// TwinCAT 3 PLC project PLC
// ProgramVersion: 3.1.4026.19
// CompilerDefines: VISU_USEPROPERTYINFO
// libraries:
//   Tc2_MC2, * (Beckhoff Automation GmbH)
//   Tc2_Standard, * (Beckhoff Automation GmbH)
//   Tc2_System, * (Beckhoff Automation GmbH)
//   VisuDialogs, * (System)
// project tree:
//   / GlobalTextList.TcGTLO, PlcTask.TcTTO, Visualization Manager.TcVMO (not stored)
//   POUs/ MAIN.TcPOU
//   VISUs/ HomeScreen.TcVIS

CONFIGURATION PLC
    RESOURCE PLC ON TwinCAT3
        TASK PlcTask(INTERVAL := T#10ms, PRIORITY := 20);
        PROGRAM MAIN WITH PlcTask : MAIN;
    END_RESOURCE
END_CONFIGURATION

// ---- POUs/MAIN.TcPOU
PROGRAM MAIN
VAR
	axisVirtualMotor : AXIS_REF;
	fbPower : MC_Power;
	fbMoveAbs : MC_MoveAbsolute;
	bEnable : BOOL;
	bMoveStart : BOOL;
	fTargetLocation : LREAL := 250.5;
	fLocation : LREAL;
END_VAR

fbPower(
	Axis := axisVirtualMotor,
	Enable := bEnable,
	Enable_Positive := bEnable,
	Enable_Negative := bEnable,
	Override := 100.0
);

fbMoveAbs(
	Axis := axisVirtualMotor,
	Execute := bMoveStart,
	Position := fTargetLocation,
	Velocity := 100.0,
	Acceleration := 100.0,
	Deceleration := 100.0,
	Jerk := 100.0
);

fLocation := axisVirtualMotor.NcToPlc.ActPos;

END_PROGRAM

// ---- GlobalTextList.TcGTLO
TEXTLIST GlobalTextList
  621 = 'Location: %.2f mm'
  700 = 'Power Off'
  717 = 'Power On'
  63 = 'Start to Move'
  985 = 'Target: %.2f mm'
END_TEXTLIST

// ---- VISUs/HomeScreen.TcVIS
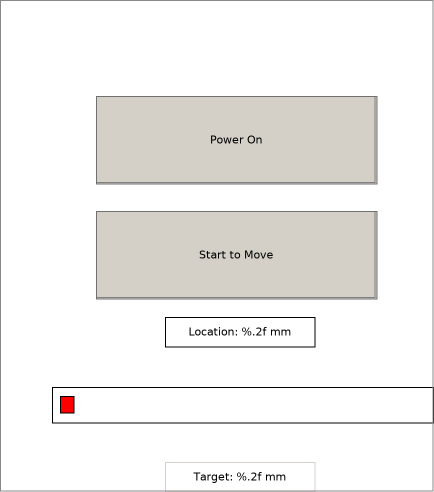
VISUALIZATION HomeScreen  // 434x492
    Button (96,96 281x88), "Power On"
        toggle MAIN.bEnable
    Button (96,211 281x88), "Start to Move"
        toggle MAIN.bMoveStart
    Rectangle (165,317 150x30), "Location: %.2f mm", text variable: MAIN.fLocation
    Textfield (165,462 150x30), "Target: %.2f mm", text variable: MAIN.fTargetLocation
        OnMouseClick: write the text variable via VisuDialogs.Numpad
    Rectangle (52,387 382x36)
    Rectangle (60,396 14x17)
        p3560616238: MAIN.fLocation
END_VISUALIZATION
